(* IEC 61131-3 sources: programs/VI-54/VI-54_20171205/VI-54_20171205/Stations/Screen/LseClass170718/Class/TitleLine, 1 file *)

(* ---- TitleLine.st ---- *)
// Eigenschaften des UDCs
//----------------------------------------------------------------------------------------------------------------------------
#define   TitleLine_UDCVersion                1           // Version des aktuellen UDCs
#define   TitleLine_VariableNo                6           // Anzahl der Variablen, die dem UDC mitgegeben werden
#define   TitleLine_BoolNo                    1           // Anzahl der Boolschen-Variablen, die dem UDC mitgegeben werden
#define   TitleLine_TextschemeNo              1           // Anzahl der Textschemen, die dem UDC mitgegeben werden

(*!
<Class
	Name               = "TitleLine"
	Revision           = "1.1"
	RealtimeTask       = "false"
	CyclicTask         = "false"
	BackgroundTask     = "false"
	Sigmatek           = "true"
	OSInterface        = "false"
	HighPriority       = "false"
	Automatic          = "false"
	UpdateMode         = "Prescan"
	SharedCommandTable = "true"
	Objectsize         = "(536,120)">
	<Channels>
		<Client Name="ColumnChoice" Required="true" Internal="false" Comment="Bitmuster zum Enablen der Darstellung von Display-Items (Spalten)"/>
		<Client Name="coSystemLogging" Required="false" Internal="false" Comment="object channel to SystemLogging (optional)"/>
	</Channels>
	<Dependencies>
		<Files>
			<File Path=".\Class\TitleLine\Title.UDC"/>
		</Files>
	</Dependencies>
	<RevDoku>
		<Owner Company="Sigmatek"/>
		<Dokumentation Revision="1.1" Date="2016-09-07" Author="HubChr" Company="Sigmatek" Description="Bugfix: TitleLine did not work if placed in an Object (Lasal Screen Editor)"/>
		<Dokumentation Revision="1.0" Date="2016-05-11" Author="KaiAnd" Company="Sigmatek" Description="official start release"/>
		<Dokumentation Revision="0.10" Date="2015-09-29" Author="BraLis" Company="Sigmatek" Description="insert the method SystemLogging::LogEventText instead of TRACE-Messages"/>
		<Dokumentation Revision="0.9" Date="2015-09-28" Author="KruAle" Company="Sigmatek" Description="get udc-data in IF_Start."/>
		<Dokumentation Revision="0.8" Date="2015-09-25" Author="BraLis" Company="Sigmatek" Description="in IF_Start the TitleTextScheme will be get&#13;&#10;"/>
		<Dokumentation Revision="0.7" Date="2015-09-24" Author="BraLis" Company="Sigmatek" Description="changed the bit combination in the methods TableLine and DrawHeader&#13;&#10;"/>
		<Dokumentation Revision="0.6" Date="2015-09-22" Company="Sigmatek" Description="Creation."/>
	</RevDoku>
	<Network Name="TitleLine">
		<!-- List of Components in this network -->
		<Components>
			<Object
				Name       = "_base"
				Class      = "_MyIO"
				Position   = "(218,120)"
				Visualized = "true">
				<Channels>
					<Server Name="Refresh"/>
					<Server Name="Server0"/>
					<Client Name="Graphic"/>
					<Client Name="Lse"/>
				</Channels>
			</Object>
		</Components>
		<Comments>
		</Comments>
		<!-- List of Connections in this network -->
		<Connections>
			<Connection Source="this.Server0" Destination="_base.Server0" Vertices="(690,210),(518,210),"/>
			<Connection Source="this.Refresh" Destination="_base.Refresh" Vertices="(690,270),(518,270),"/>
			<Connection Source="_base.Lse" Destination="this.Lse" Vertices="(218,210),(38,210),"/>
		</Connections>
		<!-- Headerfiles -->
		<Options>
		</Options>
	</Network>
</Class>
*)
#pragma using _MyIO

TitleLine : CLASS
: _MyIO
	TYPE
#pragma pack(push, 1)
	  T_S_EXTVISPARA : STRUCT  //! <Type Public="true" Name="T_S_EXTVISPARA"/>
	    bParaVar : BOOL;
	    ParaTextscheme : _ANYTHING;
	  END_STRUCT;
#pragma pack(pop)
	END_TYPE
  //Servers:
  //Clients:
	ColumnChoice 	: CltCh_BDINT;
	coSystemLogging 	: CltChCmd_SystemLogging;
  //Variables:
		bFirstRun 	: BOOL;
		ScrollOffset 	: _KOORD;
		ExtVisPara 	: T_S_EXTVISPARA;
		bGetTheurgeData 	: BOOL;
		aColumnWidths : ARRAY [0..TitleLine_VariableNo-1] OF DINT;

		aVarSingle : ARRAY [0..TitleLine_VariableNo-1] OF _VARSINGLE;

		bInitialized 	: BOOL;
		IsCon_coSystemLogging 	: BOOL;
  //Functions:

	FUNCTION VIRTUAL GLOBAL Init;

	FUNCTION TitleLine
		VAR_OUTPUT
			ret_code 	: ConfStates;
		END_VAR;
				//! <Function Comment="this method is called everytime when system wants to redraw the io" Name="Draw"/>
	FUNCTION __CDECL VIRTUAL GLOBAL Draw
		VAR_INPUT
			pio 	: ^_IO;			//! <Variable Comment="pointer to _IO information" Name="Draw.pio"/>
			pr 	: ^_RESULT;			//! <Variable Comment="pointer to _RESULT information" Name="Draw.pr"/>
			pv 	: ^_VARIABLE;			//! <Variable Comment="pointer to io _VARIABLE information" Name="Draw.pv"/>
			input 	: BOOL;			//! <Variable Comment="TRUE it&apos;s an input&#13;&#10;FALSE it&apos;s an output" Name="Draw.input"/>
		END_VAR
		VAR_OUTPUT
			retcode (EAX) 	: _DOIT;			//! <Variable Comment="for the returnstatement there are 3 different possibilities&#13;&#10;  _IDLE ..... the system should goon like it is (system goes on)&#13;&#10;  _IDIDIT ... i did it (system is ready)&#13;&#10;  _IFAILED .. i tried to do my best, but i failed (system is re" Name="Draw.retcode"/>
		END_VAR;
				//! <Function Comment="this method is called once right in front of drawing the object.&#13;&#10;for example open screen&#13;&#10;" Name="IF_Start"/>
	FUNCTION __CDECL VIRTUAL GLOBAL IF_Start
		VAR_INPUT
			pio 	: ^_IO;			//! <Variable Comment="pointer to _IO information" Name="IF_Start.pio"/>
			firsttime 	: BOOL;			//! <Variable Comment="true: when system wants to view drawing after open screen&#13;&#10;false: when system wants to redraw background" Name="IF_Start.firsttime"/>
		END_VAR;
				//! <Function Comment="method is called cyclic during object is on screen&#13;&#10;&#13;&#10;pio ....... &#13;&#10;input .... TRUE it&apos;s an input / FALSE it&apos;s an output&#13;&#10;" Name="IF_Run"/>
	FUNCTION __CDECL VIRTUAL GLOBAL IF_Run
		VAR_INPUT
			pio 	: ^_IO;			//! <Variable Comment="pointer to _IO information given by LSE" Name="IF_Run.pio"/>
			input 	: BOOL;			//! <Variable Comment="TRUE it&apos;s an input&#13;&#10;FALSE it&apos;s an output" Name="IF_Run.input"/>
		END_VAR;

	FUNCTION VIRTUAL TableLines
		VAR_INPUT
			pio 	: ^_IO;
		END_VAR
		VAR_OUTPUT
			bSuccessful 	: BOOL;
		END_VAR;

	FUNCTION VIRTUAL DrawHeader
		VAR_INPUT
			pio 	: ^_IO;
		END_VAR
		VAR_OUTPUT
			bSuccessful 	: BOOL;
		END_VAR;

	FUNCTION GLOBAL setActLineBegin
		VAR_INPUT
			NewScrollOffset 	: _KOORD;
		END_VAR;

	FUNCTION GLOBAL GetTitleTxtScheme
		VAR_INPUT
			pTxtScheme 	: ^_ANYTHING;
		END_VAR
		VAR_OUTPUT
			RetCode 	: BOOL;
		END_VAR;

	FUNCTION GetTheUrge
		VAR_INPUT
			pio 	: ^_IO;
		END_VAR
		VAR_OUTPUT
			bSuccessful 	: BOOL;
		END_VAR;

	FUNCTION GetTheUrgeValues
		VAR_INPUT
			pio 	: ^_IO;
		END_VAR
		VAR_OUTPUT
			bSuccessful 	: BOOL;
		END_VAR;
  //Tables:
	FUNCTION @STD
		VAR_OUTPUT
			ret_code	: CONFSTATES;
		END_VAR;
	FUNCTION GLOBAL TAB @CT_;
END_CLASS;

#pragma usingLtd SystemLogging

FUNCTION VIRTUAL GLOBAL TitleLine::Init

  if (_FirstScan) then

    //-------------------------------------------------------------------------
    //  check client-connnections and set flags                   KaiAnd
    //-------------------------------------------------------------------------
    if (IsClientConnected(#coSystemLogging)) then
      IsCon_coSystemLogging := TRUE;
    else
      IsCon_coSystemLogging := FALSE;
    end_if;
    //-------------------------------------------------------------------------
  end_if;

END_FUNCTION

FUNCTION __CDECL VIRTUAL GLOBAL TitleLine::IF_Start
	VAR_INPUT
		pio 	: ^_IO;
		firsttime 	: BOOL;
	END_VAR

  // Basisklasse aufrufen
  _MyIO::IF_Start(pio:=pio, firsttime:=firsttime);

  bInitialized := GetTheUrge(pio:=pio);

  // Erster Aufruf
  //--------------------------------------------------------------------------------------------
  if bFirstRun = false then

    // erster Start ist vorbei
    bFirstRun := true;

    // Kein Scroll-Offset
    ScrollOffset := pio^.space.xy1.x + 1;  // HubChr v1.1 use pio^.space instead of pio^.room

  end_if;

END_FUNCTION

FUNCTION __CDECL VIRTUAL GLOBAL TitleLine::Draw
	VAR_INPUT
		pio 	: ^_IO;
		pr 	: ^_RESULT;
		pv 	: ^_VARIABLE;
		input 	: BOOL;
	END_VAR
	VAR_OUTPUT
		retcode (EAX) 	: _DOIT;
	END_VAR

  // UDC-Parameter schon geholt?
  if bInitialized then

    // Parameter vom UDC holen
    GetTheUrgeValues(pio:=pio);

    // Konfiguration der Spalten lesen
    ColumnChoice := ColumnChoice.Read();

    // Rahmen zeichnen
    DrawButton(#pio^.space, T_FILL or T_COPY or T_SOLID, pio^.frametype, pio^.colback, pio^.colframe); // HubChr v1.1 use pio^.space instead of pio^.room

    // Zeilenunterteilung zeichnen
    //-----------------------------------------------------------------------------------------
    if ExtVisPara.bParaVar = true then

      if TableLines(pio:=pio) = false then
        if (IsCon_coSystemLogging = True) then    // KaiAnd
          coSystemLogging.LogEventText("AlarmTitle::Draw(): Zeichnen der Kopfzeile fehlgeschlagen");
        end_if;
      end_if;

    end_if;

    // Texte in Spalten ausgeben
    //-----------------------------------------------------------------------------------------
    if DrawHeader(pio:=pio) = false then
      if (IsCon_coSystemLogging = True) then    // KaiAnd
        coSystemLogging.LogEventText("AlarmTitle::Draw(): Zeichnen der Kopfzeile fehlgeschlagen");
      end_if;
    end_if;

    // Rahmen erneut zeichnen, falls Scrollliste horizontal verschoben wurde
    DrawButton(#pio^.space, T_FILL or T_COPY or T_SOLID, pio^.frametype, INVISIBLE, pio^.colframe); // HubChr v1.1 use pio^.space instead of pio^.room

    // Rückgabewert setzen
    retcode := _IDIDIT;

  else
    retcode := _IFAILED;
  end_if;

END_FUNCTION

FUNCTION VIRTUAL TitleLine::TableLines
	VAR_INPUT
		pio 	: ^_IO;
	END_VAR
	VAR_OUTPUT
		bSuccessful 	: BOOL;
	END_VAR
  VAR
    tmpRoom   : _ROOM;
  END_VAR

  // Übergabeparameter prüfen
  if pio = NIL then
    bSuccessful := false;
    return;
  else
    bSuccessful := true;
  end_if;

  // Bereich definieren
  tmpRoom.xy1.x := ScrollOffset;
  tmpRoom.xy1.y := pio^.space.xy1.y; // HubChr v1.1 use pio^.space instead of pio^.room
  tmpRoom.xy2.x := ScrollOffset;
  tmpRoom.xy2.y := pio^.space.xy2.y; // HubChr v1.1 use pio^.space instead of pio^.room

  // Trennline zwischen Spalte1 und Spalte2
  //-----------------------------------------------------------------------------------------
  if ColumnChoice AND 2#000001 then
    // Koordinaten bestimmen
    tmpRoom.xy1.x := tmpRoom.xy2.x + to_int(aColumnWidths[0]);
    tmpRoom.xy2.x := tmpRoom.xy1.x;

    Graphic.Line( x1      := tmpRoom.xy1.x,
                  y1      := tmpRoom.xy1.y,
                  x2      := tmpRoom.xy2.x,
                  y2      := tmpRoom.xy2.y,
                  attrib  := T_SOLID,
                  color   := pio^.colframe);
  end_if;

  // Trennline zwischen Spalte2 und Spalte3
  //-----------------------------------------------------------------------------------------
  if ColumnChoice AND 2#000010 then
    // Koordinaten bestimmen
    tmpRoom.xy1.x := tmpRoom.xy2.x + to_int(aColumnWidths[1]);
    tmpRoom.xy2.x := tmpRoom.xy1.x;

    Graphic.Line( x1      := tmpRoom.xy1.x,
                  y1      := tmpRoom.xy1.y,
                  x2      := tmpRoom.xy2.x,
                  y2      := tmpRoom.xy2.y,
                  attrib  := T_SOLID,
                  color   := pio^.colframe);
  end_if;

  // Trennline zwischen Spalte3 und Spalte4
  //-----------------------------------------------------------------------------------------
  if ColumnChoice AND 2#000100 then
    // Koordinaten bestimmen
    tmpRoom.xy1.x := tmpRoom.xy2.x + to_int(aColumnWidths[2]);
    tmpRoom.xy2.x := tmpRoom.xy1.x;

    Graphic.Line( x1      := tmpRoom.xy1.x,
                  y1      := tmpRoom.xy1.y,
                  x2      := tmpRoom.xy2.x,
                  y2      := tmpRoom.xy2.y,
                  attrib  := T_SOLID,
                  color   := pio^.colframe);
  end_if;

  // Trennline zwischen Spalte4 und Spalte5
  //-----------------------------------------------------------------------------------------
  if ColumnChoice AND 2#001000 then
    // Koordinaten bestimmen
    tmpRoom.xy1.x := tmpRoom.xy2.x + to_int(aColumnWidths[3]);
    tmpRoom.xy2.x := tmpRoom.xy1.x;

    Graphic.Line( x1      := tmpRoom.xy1.x,
                  y1      := tmpRoom.xy1.y,
                  x2      := tmpRoom.xy2.x,
                  y2      := tmpRoom.xy2.y,
                  attrib  := T_SOLID,
                  color   := pio^.colframe);
  end_if;

  // Trennline zwischen Spalte5 und Spalte6
  //-----------------------------------------------------------------------------------------
  if ColumnChoice AND 2#010000 then
    // Koordinaten bestimmen
    tmpRoom.xy1.x := tmpRoom.xy2.x + to_int(aColumnWidths[4]);
    tmpRoom.xy2.x := tmpRoom.xy1.x;

    Graphic.Line( x1      := tmpRoom.xy1.x,
                  y1      := tmpRoom.xy1.y,
                  x2      := tmpRoom.xy2.x,
                  y2      := tmpRoom.xy2.y,
                  attrib  := T_SOLID,
                  color   := pio^.colframe);
  end_if;

END_FUNCTION

FUNCTION VIRTUAL TitleLine::DrawHeader
	VAR_INPUT
		pio 	: ^_IO;
	END_VAR
	VAR_OUTPUT
		bSuccessful 	: BOOL;
	END_VAR
  VAR
    pString     : ^_CHAR;
    tmpRoom     : _ROOM;
    fieldHight  : INT;
    fontWidth   : UINT;
    fontHight   : UINT;
  END_VAR

  // Übergabeparameter prüfen
  if pio = NIL then
    bSuccessful := false;
    return;
  else
    bSuccessful := true;
  end_if;

  // Bestimmen der Position des Texts (Zentriert im Feld)
  fieldHight := pio^.space.xy2.y - pio^.space.xy1.y;    // HubChr v1.1 use pio^.space instead of pio^.room
  font_size(x0:=pio^.font, p1:=#fontWidth, p2:=#fontHight);

  tmpRoom.xy1.x := ScrollOffset - 1;
  tmpRoom.xy1.y := pio^.space.xy1.y + ((fieldHight / 2) - (fontHight$INT / 2)); // HubChr v1.1 use pio^.space instead of pio^.room
  tmpRoom.xy2.x := ScrollOffset-1;
  tmpRoom.xy2.y := tmpRoom.xy1.y + fontHight$INT;

  // Prüfen ob Text der Spalte1 dargestellt werden soll
  //-----------------------------------------------------------------------------------------
  if ColumnChoice AND 2#000001 then

    // Text aus Textschema holen
    pString$^void := NewDoScheme(x0 := TEXTSCHEME,
                                 x1 := 0,
                                 x2 := ExtVisPara.ParaTextscheme.no);
    if pString = NIL then
      if (IsCon_coSystemLogging = True) then    // KaiAnd
        coSystemLogging.LogEventText("UserListTitel::DrawHeader(): Keinen Text (Eventzeit) gefunden");
      end_if;
    else
      // Koordinaten bestimmen
      tmpRoom.xy1.x := tmpRoom.xy1.x + 5;
      tmpRoom.xy2.x := tmpRoom.xy1.x + to_int(aColumnWidths[0]) - 5;

      // Text ausgeben
      OutTextAlign( p0 := pString,
                    x1 := 0,
                    p1 := #tmpRoom,
                    x2 := pio^.font,
                    x3 := pio^.attrib,
                    x9 := _DEFFRAME,
                    x4 := pio^.coltxt,
                    x5 := INVISIBLE,
                    x6 := NIL$_COLOR,
                    x7 := sizeof(_CHAR));
    end_if;

  end_if;

  // Prüfen ob Text der Spalte2 dargestellt werden soll
  //-----------------------------------------------------------------------------------------
  if ColumnChoice AND 2#000010 then

    // Text aus Textschema holen
    pString$^void := NewDoScheme(x0 := TEXTSCHEME,
                                 x1 := 1,
                                 x2 := ExtVisPara.ParaTextscheme.no);
    if pString = NIL then
      if (IsCon_coSystemLogging = True) then    // KaiAnd
        coSystemLogging.LogEventText("TitleLine::DrawHeader(): Keinen Text (Eventzeit) gefunden");
      end_if;
    else
      // Koordinaten bestimmen
      tmpRoom.xy1.x := tmpRoom.xy2.x + 5;
      tmpRoom.xy2.x := tmpRoom.xy1.x + to_int(aColumnWidths[1]) - 5;

      // Text ausgeben
      OutTextAlign( p0 := pString,
                    x1 := 0,
                    p1 := #tmpRoom,
                    x2 := pio^.font,
                    x3 := pio^.attrib,
                    x9 := _DEFFRAME,
                    x4 := pio^.coltxt,
                    x5 := INVISIBLE,
                    x6 := NIL$_COLOR,
                    x7 := sizeof(_CHAR));
    end_if;

  end_if;

  // Prüfen ob Text der Spalte3 dargestellt werden soll
  //-----------------------------------------------------------------------------------------
  if ColumnChoice AND 2#000100 then

    //Text aus Textschema holen
    pString$^void := NewDoScheme(x0 := TEXTSCHEME,
                                 x1 := 2,
                                 x2 := ExtVisPara.ParaTextscheme.no);
    if pString = NIL then
      if (IsCon_coSystemLogging = True) then    // KaiAnd
        coSystemLogging.LogEventText("TitleLine::DrawHeader(): Keinen Text (Alarmnummer) gefunden");
      end_if;
    else
      // Koordinaten bestimmen
      tmpRoom.xy1.x := tmpRoom.xy2.x + 5;
      tmpRoom.xy2.x := tmpRoom.xy1.x + to_int(aColumnWidths[2]) - 5;

      // Text ausgeben
      OutTextAlign( p0 := pString,
                    x1 := 0,
                    p1 := #tmpRoom,
                    x2 := pio^.font,
                    x3 := pio^.attrib,
                    x9 := _DEFFRAME,
                    x4 := pio^.coltxt,
                    x5 := INVISIBLE,
                    x6 := NIL$_COLOR,
                    x7 := sizeof(_CHAR));

    end_if;

  end_if;

  // Prüfen ob Text der Spalte4 dargestellt werden soll
  //-----------------------------------------------------------------------------------------
  if ColumnChoice AND 2#001000 then

    // Text aus Textschema holen
    pString$^void := NewDoScheme(x0 := TEXTSCHEME,
                                 x1 := 3,
                                 x2 := ExtVisPara.ParaTextscheme.no);
    if pString = NIL then
      if (IsCon_coSystemLogging = True) then    // KaiAnd
        coSystemLogging.LogEventText("TitleLine::DrawHeader(): Keinen Text (Accesslevel) gefunden");
      end_if;
    else
      // Koordinaten bestimmen
      tmpRoom.xy1.x := tmpRoom.xy2.x + 5;
      tmpRoom.xy2.x := tmpRoom.xy1.x + to_int(aColumnWidths[3]) - 5;

      // Text ausgeben
      OutTextAlign( p0 := pString,
                    x1 := 0,
                    p1 := #tmpRoom,
                    x2 := pio^.font,
                    x3 := pio^.attrib,
                    x9 := _DEFFRAME,
                    x4 := pio^.coltxt,
                    x5 := INVISIBLE,
                    x6 := NIL$_COLOR,
                    x7 := sizeof(_CHAR));
    end_if;

  end_if;

  // Prüfen ob Text der Spalte5 dargestellt werden soll
  //-----------------------------------------------------------------------------------------
  if ColumnChoice AND 2#010000 then

    // Text aus Textschema holen
    pString$^void := NewDoScheme(x0 := TEXTSCHEME,
                                 x1 := 4,
                                 x2 := ExtVisPara.ParaTextscheme.no);
    if pString = NIL then
      if (IsCon_coSystemLogging = True) then    // KaiAnd
        coSystemLogging.LogEventText("TitleLine::DrawHeader(): Keinen Text (Beschreibung) gefunden");
      end_if;
    else
      // Koordinaten bestimmen
      tmpRoom.xy1.x := tmpRoom.xy2.x + 5;
      tmpRoom.xy2.x := tmpRoom.xy1.x + to_int(aColumnWidths[4]) - 5;

      // Text ausgeben
      OutTextAlign( p0 := pString,
                    x1 := 0,
                    p1 := #tmpRoom,
                    x2 := pio^.font,
                    x3 := pio^.attrib,
                    x9 := _DEFFRAME,
                    x4 := pio^.coltxt,
                    x5 := INVISIBLE,
                    x6 := NIL$_COLOR,
                    x7 := sizeof(_CHAR));
    end_if;

  end_if;

  // Prüfen ob Text der Spalte6 dargestellt werden soll
  //-----------------------------------------------------------------------------------------
  if ColumnChoice AND 2#100000 then

    // Text aus Textschema holen
    pString$^void := NewDoScheme(x0 := TEXTSCHEME,
                                 x1 := 5,
                                 x2 := ExtVisPara.ParaTextscheme.no);
    if pString = NIL then
      if (IsCon_coSystemLogging = True) then    // KaiAnd
        coSystemLogging.LogEventText("TitleLine::DrawHeader(): Keinen Text (Beschreibung) gefunden");
      end_if;
    else
      // Koordinaten bestimmen
      tmpRoom.xy1.x := tmpRoom.xy2.x + 5;
      tmpRoom.xy2.x := tmpRoom.xy1.x + to_int(aColumnWidths[5]) - 5;

      // Text ausgeben
      OutTextAlign( p0 := pString,
                    x1 := 0,
                    p1 := #tmpRoom,
                    x2 := pio^.font,
                    x3 := T_LEFTBOUND or T_SOLID or T_PROP or T_COPY or T_MIDBOUND,
                    x9 := _DEFFRAME,
                    x4 := pio^.coltxt,
                    x5 := INVISIBLE,
                    x6 := NIL$_COLOR,
                    x7 := sizeof(_CHAR));
    end_if;

  end_if;

END_FUNCTION

FUNCTION __CDECL VIRTUAL GLOBAL TitleLine::IF_Run
	VAR_INPUT
		pio 	: ^_IO;
		input 	: BOOL;
	END_VAR

  // Spalten ab/angewählt?
  //-----------------------------------------------------------------------------------------
  if ColumnChoice <> ColumnChoice.Read() then

    // Neue Konfiguration speichern
    ColumnChoice := ColumnChoice.Read();

    // Kopfzeile neu zeichnen
    Refresh.Write(1);

  end_if;

END_FUNCTION

FUNCTION GLOBAL TitleLine::setActLineBegin
	VAR_INPUT
		NewScrollOffset 	: _KOORD;
	END_VAR

  // Hat sich der Offset verändert?
  //-----------------------------------------------------------------------------------------
  if ScrollOffset <> NewScrollOffset then

    // Neuen Offset speichern
    ScrollOffset := NewScrollOffset;

    // Kopfzeile neu zeichnen
    Refresh.Write(1);

  end_if;

END_FUNCTION

FUNCTION GLOBAL TitleLine::GetTitleTxtScheme
	VAR_INPUT
		pTxtScheme 	: ^_ANYTHING;
	END_VAR
	VAR_OUTPUT
		RetCode 	: BOOL;
	END_VAR

  RetCode := false;

  if pTxtScheme <> NIL then

    if bGetTheurgeData = true then
      pTxtScheme^ := ExtVisPara.ParaTextscheme;
      RetCode := true;
    end_if;

  end_if;

END_FUNCTION

FUNCTION TitleLine::GetTheUrge
	VAR_INPUT
		pio 	: ^_IO;
	END_VAR
	VAR_OUTPUT
		bSuccessful 	: BOOL;
	END_VAR
  VAR
    tmpCounter      : UINT;
    pBool           : ^BOOL;
    pHelpAnyThing   : ^_ANYTHING;
	  pVarLabel       : ^_VARLABEL;
  END_VAR

  // Gültiger Übergabeparameter?
  if (pio <> NIL) & (pio^.theurge <> NIL) then

    // Richtige Version des UDCs?
    if (pio^.theurge^.info = TitleLine_UDCVersion) then

      bSuccessful := true;

      // Boolparameter holen
      //-----------------------------------------------------------------------------------------
      if pio^.theurge^.membool.no = TitleLine_BoolNo then

        pBool := pio^.theurge^.membool.ptr;
        ExtVisPara.bParaVar := pBool^$USINT;

      else
        bSuccessful := false;
      end_if;

      // Index des Textschemas holen
      //-----------------------------------------------------------------------------------------
      if (pio^.theurge^.memanything.no = TitleLine_TextschemeNo) then

        pHelpAnyThing := pio^.theurge^.memanything.ptr;

        // Schema ein Textschema?
        if (pHelpAnyThing^.list = TEXTSCHEME) then
          ExtVisPara.ParaTextscheme.list := pHelpAnyThing^.list;
          ExtVisPara.ParaTextscheme.no   := pHelpAnyThing^.no;
        else
          ExtVisPara.ParaTextscheme.list := DEFLST;
          ExtVisPara.ParaTextscheme.no   := DEFSCOPE;
          if (IsCon_coSystemLogging = True) then    // KaiAnd
            coSystemLogging.LogEventText("TitleLine::GetFirstTheUrge(): Verweis auf Textliste konnte nicht bestimmt werden");
          end_if;
        end_if;

      else
        bSuccessful := false;
      end_if;

      // variable informations
      //--------------------------------------------------------------
      // check number of variables
      if pio^.theurge^.memvarlabel.no = TitleLine_VariableNo then

        // pointer to variable informations
        pVarLabel := pio^.theurge^.memvarlabel.ptr;

        // loop to store all parameter
        for tmpCounter:=0 to sizeof(aVarSingle) / sizeof(aVarSingle[0]) - 1 do

          // save variable informations
          aVarSingle[tmpCounter] := pVarLabel^.info[0];

          // check for constant
          if aVarSingle[tmpCounter].state = CONST_VAL then
            aColumnWidths[tmpCounter] := aVarSingle[tmpCounter].value;
          end_if;

          // step to next variable
          pVarLabel += sizeof(_VARLABEL);

        end_for;

      else
        bSuccessful := false;
      end_if;

      bGetTheurgeData := true; // RauAnd : es wurden das erste mal die Einträge aus dem UDC geholt.

    else
      bSuccessful := false;
      if (IsCon_coSystemLogging = True) then    // KaiAnd
        coSystemLogging.LogEventText("TitleLine::GetTheUrge(): Falsche Version des UDCs");
      end_if;
    end_if;

  else
    bSuccessful := false;
   if (IsCon_coSystemLogging = True) then    // KaiAnd
      coSystemLogging.LogEventText("TitleLine::GetTheUrge(): Ungültiger Übergabeparameter");
   end_if;
  end_if;

END_FUNCTION

FUNCTION TitleLine::GetTheUrgeValues
	VAR_INPUT
		pio 	: ^_IO;
	END_VAR
	VAR_OUTPUT
		bSuccessful 	: BOOL;
	END_VAR
  VAR
    tmpCounter  : USINT;
    tmpResult   : _RESULT;
    tmpVariable : _VARIABLE;
    tmpVarLabel : _VARLABEL;
  END_VAR

  bSuccessful := true;

  // loop to check all variables
  for tmpCounter := 0 to sizeof(aVarSingle) / sizeof(aVarSingle[0]) - 1 do

    // check if variable is a dataserver
    if aVarSingle[tmpCounter].state = VAR_VAL then

      // build varlabel
      tmpVarLabel.no      := 1;
      tmpVarLabel.info[0] := aVarSingle[tmpCounter];

      // get server-value
      if VarList_GetSystemData( p0  := #tmpResult,
                                p1  := #tmpVariable,
                                p2  := #tmpVarLabel,
                                x3  := false) = true then

        // save the new value + change checksum
        aColumnWidths[tmpCounter] := tmpResult.value;

      else
        bSuccessful := false;
      end_if;

    end_if;

  end_for;

END_FUNCTION

FUNCTION TitleLine::TitleLine
	VAR_OUTPUT
		ret_code 	: ConfStates;
	END_VAR

	ret_code := C_OK;

END_FUNCTION
